{attribute addProperty BoxType "KL1862"}
{attribute addProperty Id "Channel_1Channel_70B606D100Channel_2Channel_70B606D100Channel_3Channel_70B606D100Channel_4Channel_70B606D100Channel_5Channel_70B606D100Channel_6Channel_70B606D100Channel_7Channel_70B606D100Channel_8Channel_70B606D100Channel_9Channel_70B606D100Channel_10Channel_70B606D100Channel_11Channel_70B606D100Channel_12Channel_70B606D100Channel_13Channel_70B606D100Channel_14Channel_70B606D100Channel_15Channel_70B606D100Channel_16Channel_70B606D100"}
{attribute addProperty CRC "2979952422"}
{attribute addProperty SizeInBites "0"}
{attribute addProperty SizeInBytes "0"}
TYPE KL1862_B19E7726 :
STRUCT
	{attribute addProperty Name "Channel_1"}
	Channel_1 : Channel_70B606D1;
	{attribute addProperty Name "Channel_2"}
	Channel_2 : Channel_70B606D1;
	{attribute addProperty Name "Channel_3"}
	Channel_3 : Channel_70B606D1;
	{attribute addProperty Name "Channel_4"}
	Channel_4 : Channel_70B606D1;
	{attribute addProperty Name "Channel_5"}
	Channel_5 : Channel_70B606D1;
	{attribute addProperty Name "Channel_6"}
	Channel_6 : Channel_70B606D1;
	{attribute addProperty Name "Channel_7"}
	Channel_7 : Channel_70B606D1;
	{attribute addProperty Name "Channel_8"}
	Channel_8 : Channel_70B606D1;
	{attribute addProperty Name "Channel_9"}
	Channel_9 : Channel_70B606D1;
	{attribute addProperty Name "Channel_10"}
	Channel_10 : Channel_70B606D1;
	{attribute addProperty Name "Channel_11"}
	Channel_11 : Channel_70B606D1;
	{attribute addProperty Name "Channel_12"}
	Channel_12 : Channel_70B606D1;
	{attribute addProperty Name "Channel_13"}
	Channel_13 : Channel_70B606D1;
	{attribute addProperty Name "Channel_14"}
	Channel_14 : Channel_70B606D1;
	{attribute addProperty Name "Channel_15"}
	Channel_15 : Channel_70B606D1;
	{attribute addProperty Name "Channel_16"}
	Channel_16 : Channel_70B606D1;
END_STRUCT
END_TYPE

(* stored: Version 1.2.0.0, ProductVersion 3.1.4024.9
   DUT KL1862_B19E7726: Id {a4863960-7984-4f59-bbd1-4c274aee9d4f} *)
